FUNCTION_BLOCK DIO_IN_8CH (* Service Interface Function Block Type *)
  (* Standard: 61499-2 *)
  (* Version 0.0, 07/06/2021, josef, nxtControl GmBH, template *)
  PACKAGE Flexbridge.Iceblock;
  (* Compiler Cpp nxtControl builtin 1.0 *)
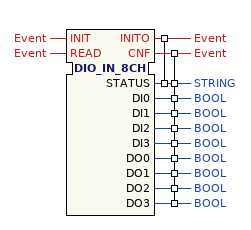
  EVENT_INPUT
    INIT;
    READ;
  END_EVENT
  EVENT_OUTPUT
    INITO WITH STATUS;
    CNF WITH STATUS, DI0, DI1, DI2, DI3, DO0, DO1, DO2, DO3;
  END_EVENT
  VAR_OUTPUT
    STATUS : STRING;
    DI0 : BOOL;
    DI1 : BOOL;
    DI2 : BOOL;
    DI3 : BOOL;
    DO0 : BOOL;
    DO1 : BOOL;
    DO2 : BOOL;
    DO3 : BOOL;
  END_VAR
  SERVICE DIO_IN_8CH/RESOURCE
    SEQUENCE normal_establishment
      DIO_IN_8CH.INIT+(PARAMS) -> RESOURCE.initialize(PARAMS) -> DIO_IN_8CH.INITO+();
    END_SEQUENCE
    SEQUENCE unsuccessful_establishment
      DIO_IN_8CH.INIT+(PARAMS) -> RESOURCE.initialize(PARAMS) -> DIO_IN_8CH.INITO-(STATUS);
    END_SEQUENCE
    SEQUENCE request_confirm
      DIO_IN_8CH.REQ+(SD) -> RESOURCE.request(SD) -> DIO_IN_8CH.CNF+(RD);
    END_SEQUENCE
    SEQUENCE request_inhibited
      DIO_IN_8CH.REQ-(SD) -> DIO_IN_8CH.CNF-(STATUS);
    END_SEQUENCE
    SEQUENCE request_error
      DIO_IN_8CH.REQ+(SD) -> RESOURCE.request(SD) -> DIO_IN_8CH.CNF-(STATUS);
    END_SEQUENCE
    SEQUENCE indication_response
      RESOURCE.indicate(RD) -> DIO_IN_8CH.IND+(RD);
      DIO_IN_8CH.RSP(QI,SD) -> RESOURCE.response(QI,SD);
    END_SEQUENCE
    SEQUENCE indication_inhibited
      RESOURCE.indicate(RD,QI=FALSE) -> RESOURCE.inhibited();
    END_SEQUENCE
    SEQUENCE error_indication
      RESOURCE.error(STATUS) -> DIO_IN_8CH.IND-(STATUS);
    END_SEQUENCE
    SEQUENCE application_initiated_termination
      DIO_IN_8CH.INIT-() -> RESOURCE.terminate() -> DIO_IN_8CH.INITO-(STATUS);
    END_SEQUENCE
    SEQUENCE resource_initiated_termination
      -> DIO_IN_8CH.INITO-(STATUS);
    END_SEQUENCE
  END_SERVICE
END_FUNCTION_BLOCK
